{attribute 'qualified_only'}
{attribute 'strict'}
TYPE E_StewartStatus :
(
	SYSTEM_OK 		:= 16#00000000,
	WARNING		 	:= 16#00000040,
	ERROR		 	:= 16#00000080
) UDINT;
END_TYPE

(* stored: Version 1.1.0.1, ProductVersion 3.1.4022.18
   DUT E_StewartStatus: Id {7a7e46e3-59f5-46d7-b122-01aa70980d96} *)
